FUNCTION_BLOCK DPFServer (* Stores 1-min resolved data for 1 day and sends it over a network upon request. Wrapper for a SERVER function block. *)
  (* Standard: 61499-2; Description: A client can request measurements (averaged since the last request) and diagnostic data from this function block. *)
  (* Version 1.0, 2017-08-27, Marc Jakobi, HTW Berlin *)
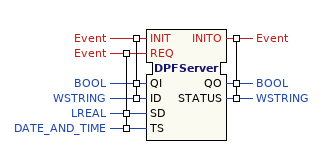
  EVENT_INPUT
    INIT WITH ID, QI; (* Initialization Request *)
    REQ WITH SD, TS; (* Normal Execution Request *)
  END_EVENT
  EVENT_OUTPUT
    INITO WITH QO, STATUS; (* Initialization Confirm *)
  END_EVENT
  VAR_INPUT
    QI : BOOL; (* Input qualifier *)
    ID : WSTRING; (* Connection identifier *)
    SD : LREAL; (* Input data *)
    TS : DATE_AND_TIME; (* Time stamp *)
  END_VAR
  VAR_OUTPUT
    QO : BOOL; (* Output event qualifier *)
    STATUS : WSTRING; (* Service status *)
  END_VAR
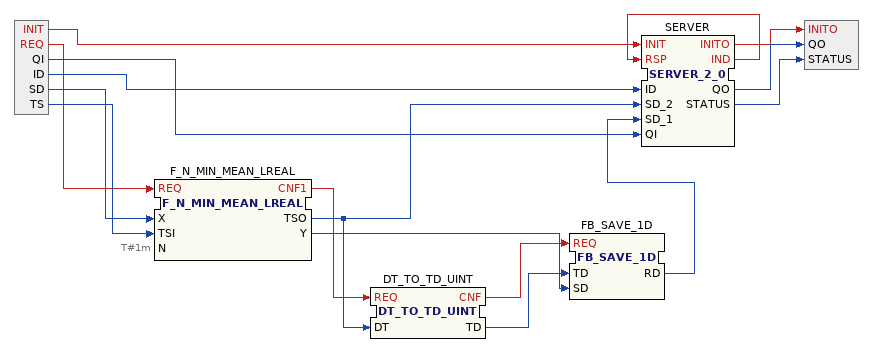
  FBS
    F_N_MIN_MEAN_LREAL : F_N_MIN_MEAN_LREAL(N := T#1m);
    DT_TO_TD_UINT : DT_TO_TD_UINT;
    SERVER : SERVER_2_0;
    FB_SAVE_1D : FB_SAVE_1D;
  END_FBS
  EVENT_CONNECTIONS
    REQ TO F_N_MIN_MEAN_LREAL.REQ;
    F_N_MIN_MEAN_LREAL.CNF1 TO DT_TO_TD_UINT.REQ;
    INIT TO SERVER.INIT;
    SERVER.INITO TO INITO;
    DT_TO_TD_UINT.CNF TO FB_SAVE_1D.REQ;
    SERVER.IND TO SERVER.RSP;
  END_CONNECTIONS
  DATA_CONNECTIONS
    SD TO F_N_MIN_MEAN_LREAL.X;
    TS TO F_N_MIN_MEAN_LREAL.TSI;
    F_N_MIN_MEAN_LREAL.TSO TO DT_TO_TD_UINT.DT;
    ID TO SERVER.ID;
    SERVER.QO TO QO;
    SERVER.STATUS TO STATUS;
    F_N_MIN_MEAN_LREAL.TSO TO SERVER.SD_2;
    DT_TO_TD_UINT.TD TO FB_SAVE_1D.TD;
    F_N_MIN_MEAN_LREAL.Y TO FB_SAVE_1D.SD;
    FB_SAVE_1D.RD TO SERVER.SD_1;
    QI TO SERVER.QI;
  END_CONNECTIONS
END_FUNCTION_BLOCK
